LIN {X 0,Y 69.281,Z 314.928,A -85,B 0,C 180,E1 -28344.379,E2 -28344.379} C_VEL
LIN {X 0,Y 66.188,Z 315.169,A -85,B 0,C 180,E1 -28352.361,E2 -28352.361} C_VEL
LIN {X 0,Y 64.354,Z 314.872,A -85,B 0,C 180,E1 -28359.206,E2 -28359.206} C_VEL
LIN {X 0,Y 64.263,Z 314.308,A -85,B 0,C 180,E1 -28364.501,E2 -28364.501} C_VEL
LIN {X 0,Y 64.59,Z 313.988,A -85,B 0,C 180,E1 -28366.232,E2 -28366.232} C_VEL
LIN {X 0,Y 67.401,Z 312.213,A -85,B 0,C 180,E1 -28374.652,E2 -28374.652} C_VEL
LIN {X 0,Y 71.651,Z 309.343,A -85,B 0,C 180,E1 -28382.65,E2 -28382.65} C_VEL
LIN {X 0,Y 77.01,Z 305.448,A -85,B 0,C 180,E1 -28389.706,E2 -28389.706} C_VEL
LIN {X 0,Y 83.494,Z 300.415,A -85,B 0,C 180,E1 -28395.684,E2 -28395.684} C_VEL
LIN {X 0,Y 90.633,Z 294.076,A -85,B 0,C 180,E1 -28400.846,E2 -28400.846} C_VEL
LIN {X 0,Y 98.27,Z 286.156,A -85,B 0,C 180,E1 -28405.328,E2 -28405.328} C_VEL
LIN {X 0,Y 99.207,Z 284.697,A -85,B 0,C 180,E1 -28406.345,E2 -28406.345} C_VEL
LIN {X 0,Y 99.897,Z 283.172,A -85,B 0,C 180,E1 -28407.591,E2 -28407.591} C_VEL
LIN {X 0,Y 100.76,Z 279.934,A -85,B 0,C 180,E1 -28410.774,E2 -28410.774} C_VEL
LIN {X 0,Y 101.285,Z 275.871,A -85,B 0,C 180,E1 -28415.397,E2 -28415.397} C_VEL
LIN {X 0,Y 101.239,Z 272.91,A -85,B 0,C 180,E1 -28419.69,E2 -28419.69} C_VEL
LIN {X 0,Y 100.997,Z 270.647,A -85,B 0,C 180,E1 -28423.838,E2 -28423.838} C_VEL
LIN {X 0,Y 100.854,Z 268.882,A -85,B 0,C 180,E1 -28427.933,E2 -28427.933} C_VEL
LIN {X 0,Y 100.705,Z 267.66,A -85,B 0,C 180,E1 -28431.976,E2 -28431.976} C_VEL
LIN {X 0,Y 101.085,Z 266.25,A -85,B 0,C 180,E1 -28440,E2 -28440} C_VEL
LIN {X 0,Y 100.934,Z 268.18,A -85,B 0,C 180,E1 -28448.005,E2 -28448.005} C_VEL
LIN {X 0,Y 100.985,Z 270.458,A -85,B 0,C 180,E1 -28453.009,E2 -28453.009} C_VEL
LIN {X 0,Y 100.891,Z 273.868,A -85,B 0,C 180,E1 -28458.268,E2 -28458.268} C_VEL
LIN {X 0,Y 100.543,Z 277.522,A -85,B 0,C 180,E1 -28462.697,E2 -28462.697} C_VEL
LIN {X 0,Y 99.953,Z 281.758,A -85,B 0,C 180,E1 -28467.196,E2 -28467.196} C_VEL
LIN {X 0,Y 99.479,Z 284.247,A -85,B 0,C 180,E1 -28469.639,E2 -28469.639} C_VEL
LIN {X 0,Y 96.47,Z 289.372,A -85,B 0,C 180,E1 -28473.09,E2 -28473.09} C_VEL
LIN {X 0,Y 94.491,Z 292.269,A -85,B 0,C 180,E1 -28475.098,E2 -28475.098} C_VEL
LIN {X 0,Y 86.974,Z 299.696,A -85,B 0,C 180,E1 -28479.855,E2 -28479.855} C_VEL
LIN {X 0,Y 80.178,Z 305.666,A -85,B 0,C 180,E1 -28485.472,E2 -28485.472} C_VEL
LIN {X 0,Y 74.049,Z 310.379,A -85,B 0,C 180,E1 -28491.907,E2 -28491.907} C_VEL
LIN {X 0,Y 69,Z 313.984,A -85,B 0,C 180,E1 -28499.383,E2 -28499.383} C_VEL
LIN {X 0,Y 66.446,Z 315.847,A -85,B 0,C 180,E1 -28504.969,E2 -28504.969} C_VEL
LIN {X 0,Y 63.235,Z 318.251,A -85,B 0,C 180,E1 -28517.155,E2 -28517.155} C_VEL
LIN {X 0,Y 62.585,Z 318.865,A -85,B 0,C 180,E1 -28523.551,E2 -28523.551} C_VEL
LIN {X 0,Y 62.61,Z 319.084,A -85,B 0,C 180,E1 -28529.998,E2 -28529.998} C_VEL
LIN {X 0,Y 62.585,Z 318.848,A -85,B 0,C 180,E1 -28536.446,E2 -28536.446} C_VEL
LIN {X 0,Y 63.234,Z 318.224,A -85,B 0,C 180,E1 -28542.842,E2 -28542.842} C_VEL
LIN {X 0,Y 64.514,Z 317.21,A -85,B 0,C 180,E1 -28549.074,E2 -28549.074} C_VEL
LIN {X 0,Y 66.444,Z 315.792,A -85,B 0,C 180,E1 -28555.028,E2 -28555.028} C_VEL
LIN {X 0,Y 70.564,Z 312.831,A -85,B 0,C 180,E1 -28563.213,E2 -28563.213} C_VEL
LIN {X 0,Y 75.928,Z 308.835,A -85,B 0,C 180,E1 -28570.384,E2 -28570.384} C_VEL
LIN {X 0,Y 82.316,Z 303.761,A -85,B 0,C 180,E1 -28576.419,E2 -28576.419} C_VEL
LIN {X 0,Y 89.407,Z 297.236,A -85,B 0,C 180,E1 -28581.817,E2 -28581.817} C_VEL
LIN {X 0,Y 94.478,Z 292.065,A -85,B 0,C 180,E1 -28584.909,E2 -28584.909} C_VEL
LIN {X 0,Y 98.362,Z 286.011,A -85,B 0,C 180,E1 -28589.024,E2 -28589.024} C_VEL
LIN {X 0,Y 99.375,Z 284.107,A -85,B 0,C 180,E1 -28590.327,E2 -28590.327} C_VEL
LIN {X 0,Y 100.293,Z 278.836,A -85,B 0,C 180,E1 -28595.638,E2 -28595.638} C_VEL
LIN {X 0,Y 100.658,Z 275.358,A -85,B 0,C 180,E1 -28599.568,E2 -28599.568} C_VEL
LIN {X 0,Y 100.795,Z 273.641,A -85,B 0,C 180,E1 -28601.714,E2 -28601.714} C_VEL
LIN {X 0,Y 100.867,Z 269.735,A -85,B 0,C 180,E1 -28607.935,E2 -28607.935} C_VEL
LIN {X 0,Y 100.801,Z 267.955,A -85,B 0,C 180,E1 -28611.985,E2 -28611.985} C_VEL
LIN {X 0,Y 100.999,Z 265.946,A -85,B 0,C 180,E1 -28620,E2 -28620} C_VEL
LIN {X 0,Y 100.537,Z 267.452,A -85,B 0,C 180,E1 -28628.037,E2 -28628.037} C_VEL
LIN {X 0,Y 100.678,Z 268.755,A -85,B 0,C 180,E1 -28632.239,E2 -28632.239} C_VEL
LIN {X 0,Y 100.972,Z 271.484,A -85,B 0,C 180,E1 -28638.253,E2 -28638.253} C_VEL
LIN {X 0,Y 101.162,Z 274.398,A -85,B 0,C 180,E1 -28642.97,E2 -28642.97} C_VEL
LIN {X 0,Y 100.959,Z 277.552,A -85,B 0,C 180,E1 -28646.901,E2 -28646.901} C_VEL
LIN {X 0,Y 100.4,Z 281.102,A -85,B 0,C 180,E1 -28650.746,E2 -28650.746} C_VEL
LIN {X 0,Y 99.192,Z 284.396,A -85,B 0,C 180,E1 -28653.646,E2 -28653.646} C_VEL
LIN {X 0,Y 98.279,Z 285.853,A -85,B 0,C 180,E1 -28654.683,E2 -28654.683} C_VEL
LIN {X 0,Y 90.667,Z 293.824,A -85,B 0,C 180,E1 -28659.184,E2 -28659.184} C_VEL
LIN {X 0,Y 83.545,Z 300.222,A -85,B 0,C 180,E1 -28664.356,E2 -28664.356} C_VEL
LIN {X 0,Y 77.07,Z 305.298,A -85,B 0,C 180,E1 -28670.334,E2 -28670.334} C_VEL
LIN {X 0,Y 71.687,Z 309.231,A -85,B 0,C 180,E1 -28677.372,E2 -28677.372} C_VEL
LIN {X 0,Y 67.418,Z 312.134,A -85,B 0,C 180,E1 -28685.358,E2 -28685.358} C_VEL
LIN {X 0,Y 65.321,Z 313.516,A -85,B 0,C 180,E1 -28691.171,E2 -28691.171} C_VEL
LIN {X 0,Y 63.559,Z 314.641,A -85,B 0,C 180,E1 -28698.761,E2 -28698.761} C_VEL
LIN {X 0,Y 62.755,Z 315.321,A -85,B 0,C 180,E1 -28710.002,E2 -28710.002} C_VEL
LIN {X 0,Y 62.952,Z 315.125,A -85,B 0,C 180,E1 -28716.411,E2 -28716.411} C_VEL
LIN {X 0,Y 64.59,Z 313.988,A -85,B 0,C 180,E1 -28726.232,E2 -28726.232} C_VEL
LIN {X 0,Y 65.433,Z 313.116,A -85,B 0,C 180,E1 -28731.326,E2 -28731.326} C_VEL
LIN {X 0,Y 66.073,Z 311.171,A -85,B 0,C 180,E1 -28739.797,E2 -28739.797} C_VEL
LIN {X 0,Y 67.331,Z 309.128,A -85,B 0,C 180,E1 -28746.33,E2 -28746.33} C_VEL
LIN {X 0,Y 69.435,Z 307.235,A -85,B 0,C 180,E1 -28750.695,E2 -28750.695} C_VEL
LIN {X 0,Y 70.429,Z 306.505,A -85,B 0,C 180,E1 -28751.967,E2 -28751.967} C_VEL
LIN {X 0,Y 78.695,Z 300.627,A -85,B 0,C 180,E1 -28759.387,E2 -28759.387} C_VEL
LIN {X 0,Y 86.318,Z 294.288,A -85,B 0,C 180,E1 -28764.51,E2 -28764.51} C_VEL
LIN {X 0,Y 93.04,Z 287.838,A -85,B 0,C 180,E1 -28768.187,E2 -28768.187} C_VEL
LIN {X 0,Y 94.084,Z 286.385,A -85,B 0,C 180,E1 -28769.206,E2 -28769.206} C_VEL
LIN {X 0,Y 95.21,Z 283.449,A -85,B 0,C 180,E1 -28772.351,E2 -28772.351} C_VEL
LIN {X 0,Y 95.93,Z 280.382,A -85,B 0,C 180,E1 -28776.238,E2 -28776.238} C_VEL
LIN {X 0,Y 96.102,Z 278.815,A -85,B 0,C 180,E1 -28778.552,E2 -28778.552} C_VEL
LIN {X 0,Y 96.171,Z 276.419,A -85,B 0,C 180,E1 -28783.003,E2 -28783.003} C_VEL
LIN {X 0,Y 96.142,Z 274.594,A -85,B 0,C 180,E1 -28787.332,E2 -28787.332} C_VEL
LIN {X 0,Y 96.163,Z 273.324,A -85,B 0,C 180,E1 -28791.595,E2 -28791.595} C_VEL
LIN {X 0,Y 96.68,Z 271.872,A -85,B 0,C 180,E1 -28800,E2 -28800} C_VEL
LIN {X 0,Y 96.394,Z 272.739,A -85,B 0,C 180,E1 -28804.181,E2 -28804.181} C_VEL
LIN {X 0,Y 96.344,Z 273.942,A -85,B 0,C 180,E1 -28808.389,E2 -28808.389} C_VEL
LIN {X 0,Y 96.215,Z 275.756,A -85,B 0,C 180,E1 -28812.658,E2 -28812.658} C_VEL
LIN {X 0,Y 95.8,Z 278.757,A -85,B 0,C 180,E1 -28817.501,E2 -28817.501} C_VEL
LIN {X 0,Y 94.94,Z 283.03,A -85,B 0,C 180,E1 -28823.013,E2 -28823.013} C_VEL
LIN {X 0,Y 94.164,Z 286.139,A -85,B 0,C 180,E1 -28826.603,E2 -28826.603} C_VEL
LIN {X 0,Y 93.455,Z 287.742,A -85,B 0,C 180,E1 -28828.088,E2 -28828.088} C_VEL
LIN {X 0,Y 89.234,Z 293.419,A -85,B 0,C 180,E1 -28832.148,E2 -28832.148} C_VEL
LIN {X 0,Y 81.307,Z 300.599,A -85,B 0,C 180,E1 -28836.911,E2 -28836.911} C_VEL
LIN {X 0,Y 72.916,Z 307.143,A -85,B 0,C 180,E1 -28843.705,E2 -28843.705} C_VEL
LIN {X 0,Y 66.59,Z 311.475,A -85,B 0,C 180,E1 -28850.708,E2 -28850.708} C_VEL
LIN {X 0,Y 62.974,Z 313.771,A -85,B 0,C 180,E1 -28856.08,E2 -28856.08} C_VEL
LIN {X 0,Y 60.046,Z 315.633,A -85,B 0,C 180,E1 -28862.082,E2 -28862.082} C_VEL
LIN {X 0,Y 57.837,Z 317.035,A -85,B 0,C 180,E1 -28868.619,E2 -28868.619} C_VEL
LIN {X 0,Y 56.317,Z 318.038,A -85,B 0,C 180,E1 -28875.545,E2 -28875.545} C_VEL
LIN {X 0,Y 55.539,Z 318.652,A -85,B 0,C 180,E1 -28882.728,E2 -28882.728} C_VEL
LIN {X 0,Y 55.509,Z 318.871,A -85,B 0,C 180,E1 -28889.998,E2 -28889.998} C_VEL
LIN {X 0,Y 55.539,Z 318.635,A -85,B 0,C 180,E1 -28897.268,E2 -28897.268} C_VEL
LIN {X 0,Y 56.316,Z 318.01,A -85,B 0,C 180,E1 -28904.452,E2 -28904.452} C_VEL
LIN {X 0,Y 57.836,Z 316.996,A -85,B 0,C 180,E1 -28911.378,E2 -28911.378} C_VEL
LIN {X 0,Y 60.044,Z 315.577,A -85,B 0,C 180,E1 -28917.915,E2 -28917.915} C_VEL
LIN {X 0,Y 64.726,Z 312.617,A -85,B 0,C 180,E1 -28926.667,E2 -28926.667} C_VEL
LIN {X 0,Y 70.65,Z 308.62,A -85,B 0,C 180,E1 -28934.131,E2 -28934.131} C_VEL
LIN {X 0,Y 78.161,Z 303.03,A -85,B 0,C 180,E1 -28940.768,E2 -28940.768} C_VEL
LIN {X 0,Y 86.505,Z 295.781,A -85,B 0,C 180,E1 -28946.38,E2 -28946.38} C_VEL
LIN {X 0,Y 89.218,Z 293.211,A -85,B 0,C 180,E1 -28947.864,E2 -28947.864} C_VEL
LIN {X 0,Y 93.345,Z 287.598,A -85,B 0,C 180,E1 -28951.898,E2 -28951.898} C_VEL
LIN {X 0,Y 94.122,Z 285.742,A -85,B 0,C 180,E1 -28953.638,E2 -28953.638} C_VEL
LIN {X 0,Y 95.102,Z 281.697,A -85,B 0,C 180,E1 -28958.315,E2 -28958.315} C_VEL
LIN {X 0,Y 95.776,Z 278.217,A -85,B 0,C 180,E1 -28962.931,E2 -28962.931} C_VEL
LIN {X 0,Y 96.067,Z 275.596,A -85,B 0,C 180,E1 -28967.322,E2 -28967.322} C_VEL
LIN {X 0,Y 96.22,Z 273.733,A -85,B 0,C 180,E1 -28971.6,E2 -28971.6} C_VEL
LIN {X 0,Y 96.281,Z 272.503,A -85,B 0,C 180,E1 -28975.814,E2 -28975.814} C_VEL
LIN {X 0,Y 96.585,Z 271.605,A -85,B 0,C 180,E1 -28980,E2 -28980} C_VEL
LIN {X 0,Y 96.005,Z 273.131,A -85,B 0,C 180,E1 -28988.419,E2 -28988.419} C_VEL
LIN {X 0,Y 95.991,Z 274.397,A -85,B 0,C 180,E1 -28992.688,E2 -28992.688} C_VEL
LIN {X 0,Y 96.041,Z 276.672,A -85,B 0,C 180,E1 -28997.959,E2 -28997.959} C_VEL
LIN {X 0,Y 95.973,Z 278.608,A -85,B 0,C 180,E1 -29001.478,E2 -29001.478} C_VEL
LIN {X 0,Y 95.822,Z 280.153,A -85,B 0,C 180,E1 -29003.791,E2 -29003.791} C_VEL
LIN {X 0,Y 95.147,Z 283.132,A -85,B 0,C 180,E1 -29007.582,E2 -29007.582} C_VEL
LIN {X 0,Y 94.711,Z 284.658,A -85,B 0,C 180,E1 -29009.326,E2 -29009.326} C_VEL
LIN {X 0,Y 94.059,Z 286.09,A -85,B 0,C 180,E1 -29010.772,E2 -29010.772} C_VEL
LIN {X 0,Y 93.045,Z 287.546,A -85,B 0,C 180,E1 -29011.822,E2 -29011.822} C_VEL
LIN {X 0,Y 85.059,Z 295.201,A -85,B 0,C 180,E1 -29016.335,E2 -29016.335} C_VEL
LIN {X 0,Y 76.325,Z 302.242,A -85,B 0,C 180,E1 -29022.557,E2 -29022.557} C_VEL
LIN {X 0,Y 69.678,Z 306.925,A -85,B 0,C 180,E1 -29029.036,E2 -29029.036} C_VEL
LIN {X 0,Y 64.084,Z 310.502,A -85,B 0,C 180,E1 -29036.748,E2 -29036.748} C_VEL
LIN {X 0,Y 61.038,Z 312.347,A -85,B 0,C 180,E1 -29042.579,E2 -29042.579} C_VEL
LIN {X 0,Y 58.639,Z 313.729,A -85,B 0,C 180,E1 -29048.929,E2 -29048.929} C_VEL
LIN {X 0,Y 56.928,Z 314.712,A -85,B 0,C 180,E1 -29055.707,E2 -29055.707} C_VEL
LIN {X 0,Y 55.671,Z 315.534,A -85,B 0,C 180,E1 -29070.002,E2 -29070.002} C_VEL
LIN {X 0,Y 55.92,Z 315.337,A -85,B 0,C 180,E1 -29077.222,E2 -29077.222} C_VEL
LIN {X 0,Y 57.697,Z 314.258,A -85,B 0,C 180,E1 -29087.799,E2 -29087.799} C_VEL
LIN {X 0,Y 61.02,Z 312.425,A -85,B 0,C 180,E1 -29097.434,E2 -29097.434} C_VEL
LIN {X 0,Y 65.779,Z 309.555,A -85,B 0,C 180,E1 -29105.991,E2 -29105.991} C_VEL
LIN {X 0,Y 70.429,Z 306.505,A -85,B 0,C 180,E1 -29111.967,E2 -29111.967} C_VEL
LIN {X 0,Y 73.248,Z 304.257,A -85,B 0,C 180,E1 -29115.717,E2 -29115.717} C_VEL
LIN {X 0,Y 77.083,Z 300.21,A -85,B 0,C 180,E1 -29121.997,E2 -29121.997} C_VEL
LIN {X 0,Y 81.476,Z 295.53,A -85,B 0,C 180,E1 -29127.466,E2 -29127.466} C_VEL
LIN {X 0,Y 84.961,Z 292.254,A -85,B 0,C 180,E1 -29129.866,E2 -29129.866} C_VEL
LIN {X 0,Y 88.204,Z 289.28,A -85,B 0,C 180,E1 -29131.44,E2 -29131.44} C_VEL
LIN {X 0,Y 89.039,Z 288.193,A -85,B 0,C 180,E1 -29132.405,E2 -29132.405} C_VEL
LIN {X 0,Y 90.369,Z 284.706,A -85,B 0,C 180,E1 -29137.117,E2 -29137.117} C_VEL
LIN {X 0,Y 90.915,Z 281.96,A -85,B 0,C 180,E1 -29141.988,E2 -29141.988} C_VEL
LIN {X 0,Y 91.084,Z 280.079,A -85,B 0,C 180,E1 -29146.616,E2 -29146.616} C_VEL
LIN {X 0,Y 91.256,Z 278.71,A -85,B 0,C 180,E1 -29151.139,E2 -29151.139} C_VEL
LIN {X 0,Y 91.955,Z 277.266,A -85,B 0,C 180,E1 -29160,E2 -29160} C_VEL
LIN {X 0,Y 91.602,Z 278.147,A -85,B 0,C 180,E1 -29164.4,E2 -29164.4} C_VEL
LIN {X 0,Y 91.216,Z 280.312,A -85,B 0,C 180,E1 -29171.105,E2 -29171.105} C_VEL
LIN {X 0,Y 90.683,Z 282.756,A -85,B 0,C 180,E1 -29175.739,E2 -29175.739} C_VEL
LIN {X 0,Y 89.761,Z 285.668,A -85,B 0,C 180,E1 -29180.02,E2 -29180.02} C_VEL
LIN {X 0,Y 88.953,Z 288.097,A -85,B 0,C 180,E1 -29183.268,E2 -29183.268} C_VEL
LIN {X 0,Y 88.357,Z 289.564,A -85,B 0,C 180,E1 -29185.027,E2 -29185.027} C_VEL
LIN {X 0,Y 85.492,Z 293.197,A -85,B 0,C 180,E1 -29187.903,E2 -29187.903} C_VEL
LIN {X 0,Y 82.787,Z 295.758,A -85,B 0,C 180,E1 -29189.522,E2 -29189.522} C_VEL
LIN {X 0,Y 74.479,Z 302.483,A -85,B 0,C 180,E1 -29194.484,E2 -29194.484} C_VEL
LIN {X 0,Y 68.195,Z 306.931,A -85,B 0,C 180,E1 -29199.38,E2 -29199.38} C_VEL
LIN {X 0,Y 61.247,Z 311.262,A -85,B 0,C 180,E1 -29206.488,E2 -29206.488} C_VEL
LIN {X 0,Y 57.205,Z 313.558,A -85,B 0,C 180,E1 -29212.098,E2 -29212.098} C_VEL
LIN {X 0,Y 53.836,Z 315.419,A -85,B 0,C 180,E1 -29218.52,E2 -29218.52} C_VEL
LIN {X 0,Y 49.466,Z 317.825,A -85,B 0,C 180,E1 -29233.49,E2 -29233.49} C_VEL
LIN {X 0,Y 48.497,Z 318.439,A -85,B 0,C 180,E1 -29241.666,E2 -29241.666} C_VEL
LIN {X 0,Y 48.427,Z 318.658,A -85,B 0,C 180,E1 -29249.998,E2 -29249.998} C_VEL
LIN {X 0,Y 48.496,Z 318.421,A -85,B 0,C 180,E1 -29258.33,E2 -29258.33} C_VEL
LIN {X 0,Y 49.465,Z 317.796,A -85,B 0,C 180,E1 -29266.506,E2 -29266.506} C_VEL
LIN {X 0,Y 51.249,Z 316.781,A -85,B 0,C 180,E1 -29274.291,E2 -29274.291} C_VEL
LIN {X 0,Y 53.834,Z 315.361,A -85,B 0,C 180,E1 -29281.477,E2 -29281.477} C_VEL
LIN {X 0,Y 59.172,Z 312.402,A -85,B 0,C 180,E1 -29290.785,E2 -29290.785} C_VEL
LIN {X 0,Y 65.727,Z 308.405,A -85,B 0,C 180,E1 -29298.457,E2 -29298.457} C_VEL
LIN {X 0,Y 74.335,Z 302.424,A -85,B 0,C 180,E1 -29305.44,E2 -29305.44} C_VEL
LIN {X 0,Y 82.774,Z 295.565,A -85,B 0,C 180,E1 -29310.488,E2 -29310.488} C_VEL
LIN {X 0,Y 85.477,Z 292.984,A -85,B 0,C 180,E1 -29312.11,E2 -29312.11} C_VEL
LIN {X 0,Y 88.245,Z 289.43,A -85,B 0,C 180,E1 -29314.939,E2 -29314.939} C_VEL
LIN {X 0,Y 89.717,Z 285.402,A -85,B 0,C 180,E1 -29320.052,E2 -29320.052} C_VEL
LIN {X 0,Y 90.599,Z 282.56,A -85,B 0,C 180,E1 -29324.246,E2 -29324.246} C_VEL
LIN {X 0,Y 91.092,Z 280.138,A -85,B 0,C 180,E1 -29328.879,E2 -29328.879} C_VEL
LIN {X 0,Y 91.497,Z 277.935,A -85,B 0,C 180,E1 -29335.595,E2 -29335.595} C_VEL
LIN {X 0,Y 91.869,Z 277.014,A -85,B 0,C 180,E1 -29340,E2 -29340} C_VEL
LIN {X 0,Y 91.139,Z 278.277,A -85,B 0,C 180,E1 -29347.672,E2 -29347.672} C_VEL
LIN {X 0,Y 90.952,Z 279.882,A -85,B 0,C 180,E1 -29353.404,E2 -29353.404} C_VEL
LIN {X 0,Y 90.762,Z 281.797,A -85,B 0,C 180,E1 -29358.043,E2 -29358.043} C_VEL
LIN {X 0,Y 90.273,Z 284.494,A -85,B 0,C 180,E1 -29362.909,E2 -29362.909} C_VEL
LIN {X 0,Y 89.019,Z 287.913,A -85,B 0,C 180,E1 -29367.575,E2 -29367.575} C_VEL
LIN {X 0,Y 88.078,Z 289.136,A -85,B 0,C 180,E1 -29368.634,E2 -29368.634} C_VEL
LIN {X 0,Y 79.7,Z 296.524,A -85,B 0,C 180,E1 -29373.102,E2 -29373.102} C_VEL
LIN {X 0,Y 71.708,Z 302.457,A -85,B 0,C 180,E1 -29378.368,E2 -29378.368} C_VEL
LIN {X 0,Y 64.466,Z 307.14,A -85,B 0,C 180,E1 -29384.88,E2 -29384.88} C_VEL
LIN {X 0,Y 58.264,Z 310.717,A -85,B 0,C 180,E1 -29392.909,E2 -29392.909} C_VEL
LIN {X 0,Y 54.84,Z 312.561,A -85,B 0,C 180,E1 -29399.164,E2 -29399.164} C_VEL
LIN {X 0,Y 52.08,Z 313.943,A -85,B 0,C 180,E1 -29406.121,E2 -29406.121} C_VEL
LIN {X 0,Y 50.086,Z 314.925,A -85,B 0,C 180,E1 -29413.704,E2 -29413.704} C_VEL
LIN {X 0,Y 48.581,Z 315.746,A -85,B 0,C 180,E1 -29430.002,E2 -29430.002} C_VEL
LIN {X 0,Y 48.885,Z 315.55,A -85,B 0,C 180,E1 -29438.268,E2 -29438.268} C_VEL
LIN {X 0,Y 50.086,Z 314.963,A -85,B 0,C 180,E1 -29446.3,E2 -29446.3} C_VEL
LIN {X 0,Y 54.822,Z 312.638,A -85,B 0,C 180,E1 -29460.851,E2 -29460.851} C_VEL
LIN {X 0,Y 60.176,Z 309.767,A -85,B 0,C 180,E1 -29469.969,E2 -29469.969} C_VEL
LIN {X 0,Y 66.696,Z 305.873,A -85,B 0,C 180,E1 -29477.53,E2 -29477.53} C_VEL
LIN {X 0,Y 74.268,Z 300.839,A -85,B 0,C 180,E1 -29483.551,E2 -29483.551} C_VEL
LIN {X 0,Y 82.393,Z 294.499,A -85,B 0,C 180,E1 -29488.539,E2 -29488.539} C_VEL
LIN {X 0,Y 84.961,Z 292.254,A -85,B 0,C 180,E1 -29489.866,E2 -29489.866} C_VEL
LIN {X 0,Y 86.403,Z 290.598,A -85,B 0,C 180,E1 -29491.316,E2 -29491.316} C_VEL
LIN {X 0,Y 86.918,Z 289.295,A -85,B 0,C 180,E1 -29493.231,E2 -29493.231} C_VEL
LIN {X 0,Y 86.766,Z 288.216,A -85,B 0,C 180,E1 -29495.751,E2 -29495.751} C_VEL
LIN {X 0,Y 85.514,Z 286.072,A -85,B 0,C 180,E1 -29503.595,E2 -29503.595} C_VEL
LIN {X 0,Y 86.013,Z 283.861,A -85,B 0,C 180,E1 -29510.594,E2 -29510.594} C_VEL
LIN {X 0,Y 86.354,Z 282.947,A -85,B 0,C 180,E1 -29515.332,E2 -29515.332} C_VEL
LIN {X 0,Y 86.921,Z 282.366,A -85,B 0,C 180,E1 -29520,E2 -29520} C_VEL
LIN {X 0,Y 86.449,Z 283.276,A -85,B 0,C 180,E1 -29524.663,E2 -29524.663} C_VEL
LIN {X 0,Y 85.871,Z 285.236,A -85,B 0,C 180,E1 -29530.843,E2 -29530.843} C_VEL
LIN {X 0,Y 85.33,Z 286.863,A -85,B 0,C 180,E1 -29534.305,E2 -29534.305} C_VEL
LIN {X 0,Y 83.877,Z 290.158,A -85,B 0,C 180,E1 -29539.582,E2 -29539.582} C_VEL
LIN {X 0,Y 83.2,Z 291.569,A -85,B 0,C 180,E1 -29541.689,E2 -29541.689} C_VEL
LIN {X 0,Y 82.157,Z 292.968,A -85,B 0,C 180,E1 -29543.131,E2 -29543.131} C_VEL
LIN {X 0,Y 80.918,Z 294.302,A -85,B 0,C 180,E1 -29544.22,E2 -29544.22} C_VEL
LIN {X 0,Y 73.608,Z 300.173,A -85,B 0,C 180,E1 -29547.969,E2 -29547.969} C_VEL
LIN {X 0,Y 63.917,Z 306.719,A -85,B 0,C 180,E1 -29554.443,E2 -29554.443} C_VEL
LIN {X 0,Y 56.299,Z 311.049,A -85,B 0,C 180,E1 -29561.493,E2 -29561.493} C_VEL
LIN {X 0,Y 51.778,Z 313.345,A -85,B 0,C 180,E1 -29567.258,E2 -29567.258} C_VEL
LIN {X 0,Y 47.891,Z 315.206,A -85,B 0,C 180,E1 -29574.053,E2 -29574.053} C_VEL
LIN {X 0,Y 42.675,Z 317.611,A -85,B 0,C 180,E1 -29590.767,E2 -29590.767} C_VEL
LIN {X 0,Y 41.471,Z 318.226,A -85,B 0,C 180,E1 -29600.241,E2 -29600.241} C_VEL
LIN {X 0,Y 41.327,Z 318.445,A -85,B 0,C 180,E1 -29609.998,E2 -29609.998} C_VEL
LIN {X 0,Y 41.47,Z 318.208,A -85,B 0,C 180,E1 -29619.755,E2 -29619.755} C_VEL
LIN {X 0,Y 42.674,Z 317.582,A -85,B 0,C 180,E1 -29629.229,E2 -29629.229} C_VEL
LIN {X 0,Y 44.835,Z 316.566,A -85,B 0,C 180,E1 -29638.049,E2 -29638.049} C_VEL
LIN {X 0,Y 47.889,Z 315.146,A -85,B 0,C 180,E1 -29645.944,E2 -29645.944} C_VEL
LIN {X 0,Y 53.967,Z 312.187,A -85,B 0,C 180,E1 -29655.743,E2 -29655.743} C_VEL
LIN {X 0,Y 61.24,Z 308.19,A -85,B 0,C 180,E1 -29663.447,E2 -29663.447} C_VEL
LIN {X 0,Y 69.904,Z 302.663,A -85,B 0,C 180,E1 -29669.822,E2 -29669.822} C_VEL
LIN {X 0,Y 79.502,Z 295.349,A -85,B 0,C 180,E1 -29674.968,E2 -29674.968} C_VEL
LIN {X 0,Y 80.904,Z 294.104,A -85,B 0,C 180,E1 -29675.796,E2 -29675.796} C_VEL
LIN {X 0,Y 82.144,Z 292.749,A -85,B 0,C 180,E1 -29676.885,E2 -29676.885} C_VEL
LIN {X 0,Y 83.134,Z 291.345,A -85,B 0,C 180,E1 -29678.418,E2 -29678.418} C_VEL
LIN {X 0,Y 84.573,Z 288.214,A -85,B 0,C 180,E1 -29683.091,E2 -29683.091} C_VEL
LIN {X 0,Y 85.238,Z 286.694,A -85,B 0,C 180,E1 -29685.679,E2 -29685.679} C_VEL
LIN {X 0,Y 85.946,Z 284.477,A -85,B 0,C 180,E1 -29690.588,E2 -29690.588} C_VEL
LIN {X 0,Y 86.345,Z 283.088,A -85,B 0,C 180,E1 -29695.331,E2 -29695.331} C_VEL
LIN {X 0,Y 86.864,Z 282.129,A -85,B 0,C 180,E1 -29700,E2 -29700} C_VEL
LIN {X 0,Y 86.288,Z 282.714,A -85,B 0,C 180,E1 -29704.672,E2 -29704.672} C_VEL
LIN {X 0,Y 85.801,Z 283.991,A -85,B 0,C 180,E1 -29710.611,E2 -29710.611} C_VEL
LIN {X 0,Y 85.357,Z 286.027,A -85,B 0,C 180,E1 -29716.749,E2 -29716.749} C_VEL
LIN {X 0,Y 84.781,Z 288.07,A -85,B 0,C 180,E1 -29721.08,E2 -29721.08} C_VEL
LIN {X 0,Y 83.606,Z 290.463,A -85,B 0,C 180,E1 -29724.854,E2 -29724.854} C_VEL
LIN {X 0,Y 74.618,Z 297.848,A -85,B 0,C 180,E1 -29729.402,E2 -29729.402} C_VEL
LIN {X 0,Y 67.528,Z 302.672,A -85,B 0,C 180,E1 -29733.636,E2 -29733.636} C_VEL
LIN {X 0,Y 59.658,Z 307.355,A -85,B 0,C 180,E1 -29740.031,E2 -29740.031} C_VEL
LIN {X 0,Y 52.77,Z 310.931,A -85,B 0,C 180,E1 -29748.25,E2 -29748.25} C_VEL
LIN {X 0,Y 48.878,Z 312.775,A -85,B 0,C 180,E1 -29754.893,E2 -29754.893} C_VEL
LIN {X 0,Y 43.336,Z 315.138,A -85,B 0,C 180,E1 -29771.076,E2 -29771.076} C_VEL
LIN {X 0,Y 41.481,Z 315.959,A -85,B 0,C 180,E1 -29790.002,E2 -29790.002} C_VEL
LIN {X 0,Y 41.888,Z 315.762,A -85,B 0,C 180,E1 -29799.661,E2 -29799.661} C_VEL
LIN {X 0,Y 43.336,Z 315.175,A -85,B 0,C 180,E1 -29808.929,E2 -29808.929} C_VEL
LIN {X 0,Y 48.848,Z 312.851,A -85,B 0,C 180,E1 -29825.137,E2 -29825.137} C_VEL
LIN {X 0,Y 54.923,Z 309.979,A -85,B 0,C 180,E1 -29834.734,E2 -29834.734} C_VEL
LIN {X 0,Y 62.125,Z 306.084,A -85,B 0,C 180,E1 -29842.364,E2 -29842.364} C_VEL
LIN {X 0,Y 70.282,Z 301.05,A -85,B 0,C 180,E1 -29848.211,E2 -29848.211} C_VEL
LIN {X 0,Y 78.919,Z 294.71,A -85,B 0,C 180,E1 -29852.942,E2 -29852.942} C_VEL
LIN {X 0,Y 83.648,Z 290.692,A -85,B 0,C 180,E1 -29855.159,E2 -29855.159} C_VEL
LIN {X 0,Y 84.844,Z 288.364,A -85,B 0,C 180,E1 -29858.769,E2 -29858.769} C_VEL
LIN {X 0,Y 85.514,Z 286.072,A -85,B 0,C 180,E1 -29863.595,E2 -29863.595} C_VEL
LIN {X 0,Y 85.266,Z 285.206,A -85,B 0,C 180,E1 -29867.544,E2 -29867.544} C_VEL
LIN {X 0,Y 84.458,Z 285.145,A -85,B 0,C 180,E1 -29871.551,E2 -29871.551} C_VEL
LIN {X 0,Y 82.963,Z 285.971,A -85,B 0,C 180,E1 -29876.98,E2 -29876.98} C_VEL
LIN {X 0,Y 80.91,Z 288.258,A -85,B 0,C 180,E1 -29885.347,E2 -29885.347} C_VEL
LIN {X 0,Y 80.362,Z 289.661,A -85,B 0,C 180,E1 -29890.073,E2 -29890.073} C_VEL
LIN {X 0,Y 79.544,Z 291.212,A -85,B 0,C 180,E1 -29893.612,E2 -29893.612} C_VEL
LIN {X 0,Y 77.868,Z 294.054,A -85,B 0,C 180,E1 -29898.612,E2 -29898.612} C_VEL
LIN {X 0,Y 76.707,Z 295.329,A -85,B 0,C 180,E1 -29900.092,E2 -29900.092} C_VEL
LIN {X 0,Y 67.468,Z 302.029,A -85,B 0,C 180,E1 -29904.403,E2 -29904.403} C_VEL
LIN {X 0,Y 57.295,Z 308.093,A -85,B 0,C 180,E1 -29910.832,E2 -29910.832} C_VEL
LIN {X 0,Y 49.259,Z 312.058,A -85,B 0,C 180,E1 -29918.303,E2 -29918.303} C_VEL
LIN {X 0,Y 42.32,Z 314.992,A -85,B 0,C 180,E1 -29928.37,E2 -29928.37} C_VEL
LIN {X 0,Y 36.027,Z 317.398,A -85,B 0,C 180,E1 -29947.033,E2 -29947.033} C_VEL
LIN {X 0,Y 34.492,Z 318.013,A -85,B 0,C 180,E1 -29958.24,E2 -29958.24} C_VEL
LIN {X 0,Y 34.242,Z 318.232,A -85,B 0,C 180,E1 -29969.997,E2 -29969.997} C_VEL
LIN {X 0,Y 34.492,Z 317.994,A -85,B 0,C 180,E1 -29981.754,E2 -29981.754} C_VEL
LIN {X 0,Y 36.026,Z 317.367,A -85,B 0,C 180,E1 -29992.962,E2 -29992.962} C_VEL
LIN {X 0,Y 38.685,Z 316.351,A -85,B 0,C 180,E1 -30003.023,E2 -30003.023} C_VEL
LIN {X 0,Y 42.317,Z 314.931,A -85,B 0,C 180,E1 -30011.627,E2 -30011.627} C_VEL
LIN {X 0,Y 49.256,Z 311.972,A -85,B 0,C 180,E1 -30021.695,E2 -30021.695} C_VEL
LIN {X 0,Y 57.29,Z 307.975,A -85,B 0,C 180,E1 -30029.17,E2 -30029.17} C_VEL
LIN {X 0,Y 66.634,Z 302.426,A -85,B 0,C 180,E1 -30035.152,E2 -30035.152} C_VEL
LIN {X 0,Y 76.702,Z 295.128,A -85,B 0,C 180,E1 -30039.909,E2 -30039.909} C_VEL
LIN {X 0,Y 77.828,Z 293.848,A -85,B 0,C 180,E1 -30041.467,E2 -30041.467} C_VEL
LIN {X 0,Y 79.498,Z 290.98,A -85,B 0,C 180,E1 -30046.513,E2 -30046.513} C_VEL
LIN {X 0,Y 80.253,Z 289.503,A -85,B 0,C 180,E1 -30049.913,E2 -30049.913} C_VEL
LIN {X 0,Y 80.877,Z 287.973,A -85,B 0,C 180,E1 -30055.015,E2 -30055.015} C_VEL
LIN {X 0,Y 81.527,Z 286.951,A -85,B 0,C 180,E1 -30060,E2 -30060} C_VEL
LIN {X 0,Y 80.585,Z 287.982,A -85,B 0,C 180,E1 -30067.247,E2 -30067.247} C_VEL
LIN {X 0,Y 80.387,Z 288.534,A -85,B 0,C 180,E1 -30070.07,E2 -30070.07} C_VEL
LIN {X 0,Y 79.817,Z 290.027,A -85,B 0,C 180,E1 -30075.317,E2 -30075.317} C_VEL
LIN {X 0,Y 79.407,Z 291.061,A -85,B 0,C 180,E1 -30078.046,E2 -30078.046} C_VEL
LIN {X 0,Y 78.643,Z 292.489,A -85,B 0,C 180,E1 -30080.945,E2 -30080.945} C_VEL
LIN {X 0,Y 75.969,Z 294.686,A -85,B 0,C 180,E1 -30082.319,E2 -30082.319} C_VEL
LIN {X 0,Y 66.846,Z 301.081,A -85,B 0,C 180,E1 -30086.666,E2 -30086.666} C_VEL
LIN {X 0,Y 58.096,Z 306.156,A -85,B 0,C 180,E1 -30092.137,E2 -30092.137} C_VEL
LIN {X 0,Y 50.162,Z 310.088,A -85,B 0,C 180,E1 -30099.597,E2 -30099.597} C_VEL
LIN {X 0,Y 43.254,Z 312.989,A -85,B 0,C 180,E1 -30109.467,E2 -30109.467} C_VEL
LIN {X 0,Y 36.696,Z 315.351,A -85,B 0,C 180,E1 -30127.481,E2 -30127.481} C_VEL
LIN {X 0,Y 34.4,Z 316.172,A -85,B 0,C 180,E1 -30150.003,E2 -30150.003} C_VEL
LIN {X 0,Y 34.92,Z 315.975,A -85,B 0,C 180,E1 -30161.614,E2 -30161.614} C_VEL
LIN {X 0,Y 36.696,Z 315.388,A -85,B 0,C 180,E1 -30172.525,E2 -30172.525} C_VEL
LIN {X 0,Y 43.229,Z 313.063,A -85,B 0,C 180,E1 -30190.567,E2 -30190.567} C_VEL
LIN {X 0,Y 50.129,Z 310.192,A -85,B 0,C 180,E1 -30200.455,E2 -30200.455} C_VEL
LIN {X 0,Y 58.066,Z 306.296,A -85,B 0,C 180,E1 -30207.916,E2 -30207.916} C_VEL
LIN {X 0,Y 66.817,Z 301.261,A -85,B 0,C 180,E1 -30213.39,E2 -30213.39} C_VEL
LIN {X 0,Y 75.954,Z 294.921,A -85,B 0,C 180,E1 -30217.715,E2 -30217.715} C_VEL
LIN {X 0,Y 78.706,Z 292.677,A -85,B 0,C 180,E1 -30219.073,E2 -30219.073} C_VEL
LIN {X 0,Y 79.51,Z 291.235,A -85,B 0,C 180,E1 -30221.978,E2 -30221.978} C_VEL
LIN {X 0,Y 79.978,Z 290.048,A -85,B 0,C 180,E1 -30225.158,E2 -30225.158} C_VEL
LIN {X 0,Y 80.527,Z 288.688,A -85,B 0,C 180,E1 -30229.947,E2 -30229.947} C_VEL
LIN {X 0,Y 80.951,Z 287.753,A -85,B 0,C 180,E1 -30235.019,E2 -30235.019} C_VEL
LIN {X 0,Y 81.578,Z 287.172,A -85,B 0,C 180,E1 -30240,E2 -30240} C_VEL
LIN {X 0,Y 80.91,Z 288.258,A -85,B 0,C 180,E1 -30245.347,E2 -30245.347} C_VEL
LIN {X 0,Y 79.983,Z 289.522,A -85,B 0,C 180,E1 -30248.075,E2 -30248.075} C_VEL
LIN {X 0,Y 78.386,Z 291.295,A -85,B 0,C 180,E1 -30250.545,E2 -30250.545} C_VEL
LIN {X 0,Y 75.477,Z 294.106,A -85,B 0,C 180,E1 -30253.439,E2 -30253.439} C_VEL
LIN {X 0,Y 71.818,Z 297.137,A -85,B 0,C 180,E1 -30255.806,E2 -30255.806} C_VEL
LIN {X 0,Y 69.722,Z 298.627,A -85,B 0,C 180,E1 -30256.705,E2 -30256.705} C_VEL
LIN {X 0,Y 60.16,Z 304.6,A -85,B 0,C 180,E1 -30260.837,E2 -30260.837} C_VEL
LIN {X 0,Y 50.966,Z 309.314,A -85,B 0,C 180,E1 -30266.316,E2 -30266.316} C_VEL
LIN {X 0,Y 42.427,Z 312.919,A -85,B 0,C 180,E1 -30274.078,E2 -30274.078} C_VEL
LIN {X 0,Y 37.288,Z 314.779,A -85,B 0,C 180,E1 -30281.066,E2 -30281.066} C_VEL
LIN {X 0,Y 29.608,Z 317.184,A -85,B 0,C 180,E1 -30301.654,E2 -30301.654} C_VEL
LIN {X 0,Y 27.561,Z 317.8,A -85,B 0,C 180,E1 -30315.223,E2 -30315.223} C_VEL
LIN {X 0,Y 27.129,Z 318.019,A -85,B 0,C 180,E1 -30329.996,E2 -30329.996} C_VEL
LIN {X 0,Y 27.561,Z 317.781,A -85,B 0,C 180,E1 -30344.77,E2 -30344.77} C_VEL
LIN {X 0,Y 29.606,Z 317.154,A -85,B 0,C 180,E1 -30358.34,E2 -30358.34} C_VEL
LIN {X 0,Y 32.94,Z 316.137,A -85,B 0,C 180,E1 -30369.793,E2 -30369.793} C_VEL
LIN {X 0,Y 37.285,Z 314.717,A -85,B 0,C 180,E1 -30378.931,E2 -30378.931} C_VEL
LIN {X 0,Y 45.185,Z 311.757,A -85,B 0,C 180,E1 -30388.805,E2 -30388.805} C_VEL
LIN {X 0,Y 53.991,Z 307.761,A -85,B 0,C 180,E1 -30395.666,E2 -30395.666} C_VEL
LIN {X 0,Y 63.575,Z 302.459,A -85,B 0,C 180,E1 -30400.779,E2 -30400.779} C_VEL
LIN {X 0,Y 71.324,Z 297.326,A -85,B 0,C 180,E1 -30403.884,E2 -30403.884} C_VEL
LIN {X 0,Y 72.688,Z 296.123,A -85,B 0,C 180,E1 -30405.204,E2 -30405.204} C_VEL
LIN {X 0,Y 74.044,Z 294.292,A -85,B 0,C 180,E1 -30409.057,E2 -30409.057} C_VEL
LIN {X 0,Y 75.105,Z 292.58,A -85,B 0,C 180,E1 -30414.631,E2 -30414.631} C_VEL
LIN {X 0,Y 75.9,Z 291.5,A -85,B 0,C 180,E1 -30420,E2 -30420} C_VEL
LIN {X 0,Y 74.944,Z 292.353,A -85,B 0,C 180,E1 -30426.77,E2 -30426.77} C_VEL
LIN {X 0,Y 74.5,Z 293.114,A -85,B 0,C 180,E1 -30430.876,E2 -30430.876} C_VEL
LIN {X 0,Y 73.487,Z 294.91,A -85,B 0,C 180,E1 -30436.994,E2 -30436.994} C_VEL
LIN {X 0,Y 68.766,Z 298.278,A -85,B 0,C 180,E1 -30439.033,E2 -30439.033} C_VEL
LIN {X 0,Y 60.824,Z 303.101,A -85,B 0,C 180,E1 -30442.431,E2 -30442.431} C_VEL
LIN {X 0,Y 51.677,Z 307.784,A -85,B 0,C 180,E1 -30447.876,E2 -30447.876} C_VEL
LIN {X 0,Y 43.228,Z 311.359,A -85,B 0,C 180,E1 -30455.624,E2 -30455.624} C_VEL
LIN {X 0,Y 38.137,Z 313.203,A -85,B 0,C 180,E1 -30462.516,E2 -30462.516} C_VEL
LIN {X 0,Y 33.723,Z 314.584,A -85,B 0,C 180,E1 -30471.307,E2 -30471.307} C_VEL
LIN {X 0,Y 30.256,Z 315.565,A -85,B 0,C 180,E1 -30482.321,E2 -30482.321} C_VEL
LIN {X 0,Y 27.302,Z 316.385,A -85,B 0,C 180,E1 -30510.004,E2 -30510.004} C_VEL
LIN {X 0,Y 28,Z 316.188,A -85,B 0,C 180,E1 -30524.54,E2 -30524.54} C_VEL
LIN {X 0,Y 30.256,Z 315.601,A -85,B 0,C 180,E1 -30537.686,E2 -30537.686} C_VEL
LIN {X 0,Y 38.117,Z 313.276,A -85,B 0,C 180,E1 -30557.525,E2 -30557.525} C_VEL
LIN {X 0,Y 45.922,Z 310.405,A -85,B 0,C 180,E1 -30567.327,E2 -30567.327} C_VEL
LIN {X 0,Y 54.632,Z 306.508,A -85,B 0,C 180,E1 -30574.228,E2 -30574.228} C_VEL
LIN {X 0,Y 63.955,Z 301.473,A -85,B 0,C 180,E1 -30579.082,E2 -30579.082} C_VEL
LIN {X 0,Y 73.542,Z 295.133,A -85,B 0,C 180,E1 -30582.874,E2 -30582.874} C_VEL
LIN {X 0,Y 74.614,Z 293.26,A -85,B 0,C 180,E1 -30589.141,E2 -30589.141} C_VEL
LIN {X 0,Y 75.265,Z 292.275,A -85,B 0,C 180,E1 -30594.642,E2 -30594.642} C_VEL
LIN {X 0,Y 75.952,Z 291.702,A -85,B 0,C 180,E1 -30600,E2 -30600} C_VEL
LIN {X 0,Y 75.193,Z 292.748,A -85,B 0,C 180,E1 -30605.363,E2 -30605.363} C_VEL
LIN {X 0,Y 74.117,Z 294.45,A -85,B 0,C 180,E1 -30610.932,E2 -30610.932} C_VEL
LIN {X 0,Y 72.725,Z 296.332,A -85,B 0,C 180,E1 -30614.894,E2 -30614.894} C_VEL
LIN {X 0,Y 71.338,Z 297.513,A -85,B 0,C 180,E1 -30616.146,E2 -30616.146} C_VEL
LIN {X 0,Y 69.722,Z 298.627,A -85,B 0,C 180,E1 -30616.705,E2 -30616.705} C_VEL
LIN {X 0,Y 64.861,Z 301.68,A -85,B 0,C 180,E1 -30617.944,E2 -30617.944} C_VEL
LIN {X 0,Y 56.044,Z 306.137,A -85,B 0,C 180,E1 -30618.919,E2 -30618.919} C_VEL
LIN {X 0,Y 46.925,Z 309.844,A -85,B 0,C 180,E1 -30620.407,E2 -30620.407} C_VEL
LIN {X 0,Y 41.686,Z 311.721,A -85,B 0,C 180,E1 -30623.028,E2 -30623.028} C_VEL
LIN {X 0,Y 33.041,Z 314.565,A -85,B 0,C 180,E1 -30631.694,E2 -30631.694} C_VEL
LIN {X 0,Y 27.848,Z 315.967,A -85,B 0,C 180,E1 -30640.786,E2 -30640.786} C_VEL
LIN {X 0,Y 20.77,Z 317.587,A -85,B 0,C 180,E1 -30670.217,E2 -30670.217} C_VEL
LIN {X 0,Y 20.022,Z 317.806,A -85,B 0,C 180,E1 -30689.995,E2 -30689.995} C_VEL
LIN {X 0,Y 20.769,Z 317.567,A -85,B 0,C 180,E1 -30709.774,E2 -30709.774} C_VEL
LIN {X 0,Y 27.846,Z 315.923,A -85,B 0,C 180,E1 -30739.21,E2 -30739.21} C_VEL
LIN {X 0,Y 33.038,Z 314.502,A -85,B 0,C 180,E1 -30748.304,E2 -30748.304} C_VEL
LIN {X 0,Y 41.939,Z 311.542,A -85,B 0,C 180,E1 -30757.165,E2 -30757.165} C_VEL
LIN {X 0,Y 51.468,Z 307.546,A -85,B 0,C 180,E1 -30762.904,E2 -30762.904} C_VEL
LIN {X 0,Y 62.975,Z 301.402,A -85,B 0,C 180,E1 -30767.54,E2 -30767.54} C_VEL
LIN {X 0,Y 67.46,Z 298.59,A -85,B 0,C 180,E1 -30768.928,E2 -30768.928} C_VEL
LIN {X 0,Y 68.353,Z 297.626,A -85,B 0,C 180,E1 -30771.433,E2 -30771.433} C_VEL
LIN {X 0,Y 68.909,Z 296.922,A -85,B 0,C 180,E1 -30774.146,E2 -30774.146} C_VEL
LIN {X 0,Y 70.026,Z 295.737,A -85,B 0,C 180,E1 -30780,E2 -30780} C_VEL
LIN {X 0,Y 69.172,Z 296.333,A -85,B 0,C 180,E1 -30785.939,E2 -30785.939} C_VEL
LIN {X 0,Y 68.206,Z 297.431,A -85,B 0,C 180,E1 -30791.893,E2 -30791.893} C_VEL
LIN {X 0,Y 67.092,Z 298.287,A -85,B 0,C 180,E1 -30793.139,E2 -30793.139} C_VEL
LIN {X 0,Y 58.487,Z 303.315,A -85,B 0,C 180,E1 -30795.996,E2 -30795.996} C_VEL
LIN {X 0,Y 48.764,Z 307.998,A -85,B 0,C 180,E1 -30800.487,E2 -30800.487} C_VEL
LIN {X 0,Y 39.522,Z 311.573,A -85,B 0,C 180,E1 -30807.242,E2 -30807.242} C_VEL
LIN {X 0,Y 33.75,Z 313.416,A -85,B 0,C 180,E1 -30813.603,E2 -30813.603} C_VEL
LIN {X 0,Y 24.201,Z 315.778,A -85,B 0,C 180,E1 -30834.497,E2 -30834.497} C_VEL
LIN {X 0,Y 20.22,Z 316.598,A -85,B 0,C 180,E1 -30870.005,E2 -30870.005} C_VEL
LIN {X 0,Y 21.207,Z 316.401,A -85,B 0,C 180,E1 -30889.358,E2 -30889.358} C_VEL
LIN {X 0,Y 24.201,Z 315.813,A -85,B 0,C 180,E1 -30905.512,E2 -30905.512} C_VEL
LIN {X 0,Y 33.736,Z 313.488,A -85,B 0,C 180,E1 -30926.444,E2 -30926.444} C_VEL
LIN {X 0,Y 42.504,Z 310.617,A -85,B 0,C 180,E1 -30935.431,E2 -30935.431} C_VEL
LIN {X 0,Y 51.944,Z 306.719,A -85,B 0,C 180,E1 -30941.284,E2 -30941.284} C_VEL
LIN {X 0,Y 61.779,Z 301.684,A -85,B 0,C 180,E1 -30945.238,E2 -30945.238} C_VEL
LIN {X 0,Y 67.178,Z 298.424,A -85,B 0,C 180,E1 -30946.975,E2 -30946.975} C_VEL
LIN {X 0,Y 68.299,Z 297.576,A -85,B 0,C 180,E1 -30948.123,E2 -30948.123} C_VEL
LIN {X 0,Y 69.267,Z 296.469,A -85,B 0,C 180,E1 -30954.176,E2 -30954.176} C_VEL
LIN {X 0,Y 70.064,Z 295.927,A -85,B 0,C 180,E1 -30960,E2 -30960} C_VEL
LIN {X 0,Y 68.976,Z 297.073,A -85,B 0,C 180,E1 -30965.848,E2 -30965.848} C_VEL
LIN {X 0,Y 68.406,Z 297.784,A -85,B 0,C 180,E1 -30968.558,E2 -30968.558} C_VEL
LIN {X 0,Y 67.527,Z 298.729,A -85,B 0,C 180,E1 -30971.013,E2 -30971.013} C_VEL
LIN {X 0,Y 58.003,Z 304.387,A -85,B 0,C 180,E1 -30974.221,E2 -30974.221} C_VEL
LIN {X 0,Y 48.232,Z 309.101,A -85,B 0,C 180,E1 -30978.71,E2 -30978.71} C_VEL
LIN {X 0,Y 41.686,Z 311.721,A -85,B 0,C 180,E1 -30983.028,E2 -30983.028} C_VEL
LIN {X 0,Y 36.488,Z 313.386,A -85,B 0,C 180,E1 -30986.431,E2 -30986.431} C_VEL
LIN {X 0,Y 27.257,Z 315.502,A -85,B 0,C 180,E1 -30991.839,E2 -30991.839} C_VEL
LIN {X 0,Y 20.037,Z 316.626,A -85,B 0,C 180,E1 -30999.513,E2 -30999.513} C_VEL
LIN {X 0,Y 15.576,Z 317.193,A -85,B 0,C 180,E1 -31012.003,E2 -31012.003} C_VEL
LIN {X 0,Y 14.532,Z 317.321,A -85,B 0,C 180,E1 -31018.342,E2 -31018.342} C_VEL
LIN {X 0,Y 12.929,Z 317.593,A -85,B 0,C 180,E1 -31049.992,E2 -31049.992} C_VEL
LIN {X 0,Y 14.272,Z 317.353,A -85,B 0,C 180,E1 -31079.492,E2 -31079.492} C_VEL
LIN {X 0,Y 18.35,Z 316.725,A -85,B 0,C 180,E1 -31099.986,E2 -31099.986} C_VEL
LIN {X 0,Y 23.806,Z 315.708,A -85,B 0,C 180,E1 -31112.323,E2 -31112.323} C_VEL
LIN {X 0,Y 29.911,Z 314.287,A -85,B 0,C 180,E1 -31120.015,E2 -31120.015} C_VEL
LIN {X 0,Y 39.72,Z 311.327,A -85,B 0,C 180,E1 -31126.685,E2 -31126.685} C_VEL
LIN {X 0,Y 49.842,Z 307.331,A -85,B 0,C 180,E1 -31130.749,E2 -31130.749} C_VEL
LIN {X 0,Y 60.106,Z 302.193,A -85,B 0,C 180,E1 -31133.608,E2 -31133.608} C_VEL
LIN {X 0,Y 62.977,Z 300.38,A -85,B 0,C 180,E1 -31135.76,E2 -31135.76} C_VEL
LIN {X 0,Y 63.812,Z 299.661,A -85,B 0,C 180,E1 -31140,E2 -31140} C_VEL
LIN {X 0,Y 63.047,Z 300.074,A -85,B 0,C 180,E1 -31145.15,E2 -31145.15} C_VEL
LIN {X 0,Y 62.845,Z 300.228,A -85,B 0,C 180,E1 -31146.421,E2 -31146.421} C_VEL
LIN {X 0,Y 59.979,Z 301.935,A -85,B 0,C 180,E1 -31148.396,E2 -31148.396} C_VEL
LIN {X 0,Y 50.129,Z 306.798,A -85,B 0,C 180,E1 -31151.083,E2 -31151.083} C_VEL
LIN {X 0,Y 40.089,Z 310.731,A -85,B 0,C 180,E1 -31155.388,E2 -31155.388} C_VEL
LIN {X 0,Y 30.406,Z 313.63,A -85,B 0,C 180,E1 -31162.409,E2 -31162.409} C_VEL
LIN {X 0,Y 18.887,Z 315.991,A -85,B 0,C 180,E1 -31181.917,E2 -31181.917} C_VEL
LIN {X 0,Y 13.132,Z 316.81,A -85,B 0,C 180,E1 -31230.008,E2 -31230.008} C_VEL
LIN {X 0,Y 14.714,Z 316.613,A -85,B 0,C 180,E1 -31258.539,E2 -31258.539} C_VEL
LIN {X 0,Y 18.889,Z 316.026,A -85,B 0,C 180,E1 -31278.094,E2 -31278.094} C_VEL
LIN {X 0,Y 30.391,Z 313.7,A -85,B 0,C 180,E1 -31297.678,E2 -31297.678} C_VEL
LIN {X 0,Y 40.073,Z 310.83,A -85,B 0,C 180,E1 -31304.718,E2 -31304.718} C_VEL
LIN {X 0,Y 50.123,Z 306.93,A -85,B 0,C 180,E1 -31308.975,E2 -31308.975} C_VEL
LIN {X 0,Y 60.013,Z 302.079,A -85,B 0,C 180,E1 -31311.678,E2 -31311.678} C_VEL
LIN {X 0,Y 62.93,Z 300.362,A -85,B 0,C 180,E1 -31313.588,E2 -31313.588} C_VEL
LIN {X 0,Y 63.394,Z 300.034,A -85,B 0,C 180,E1 -31316.182,E2 -31316.182} C_VEL
LIN {X 0,Y 63.868,Z 299.808,A -85,B 0,C 180,E1 -31320,E2 -31320} C_VEL
LIN {X 0,Y 63.021,Z 300.538,A -85,B 0,C 180,E1 -31324.324,E2 -31324.324} C_VEL
LIN {X 0,Y 60.11,Z 302.354,A -85,B 0,C 180,E1 -31326.396,E2 -31326.396} C_VEL
LIN {X 0,Y 49.847,Z 307.456,A -85,B 0,C 180,E1 -31329.259,E2 -31329.259} C_VEL
LIN {X 0,Y 38.757,Z 311.731,A -85,B 0,C 180,E1 -31333.816,E2 -31333.816} C_VEL
LIN {X 0,Y 29.915,Z 314.352,A -85,B 0,C 180,E1 -31339.984,E2 -31339.984} C_VEL
LIN {X 0,Y 23.809,Z 315.753,A -85,B 0,C 180,E1 -31347.673,E2 -31347.673} C_VEL
LIN {X 0,Y 14.532,Z 317.321,A -85,B 0,C 180,E1 -31378.342,E2 -31378.342} C_VEL
LIN {X 0,Y 12.843,Z 317.572,A -85,B 0,C 180,E1 -31393.19,E2 -31393.19} C_VEL
LIN {X 0,Y 11.168,Z 317.636,A -85,B 0,C 180,E1 -31420.614,E2 -31420.614} C_VEL
LIN {X 0,Y 13.452,Z 317.001,A -85,B 0,C 180,E1 -31467.467,E2 -31467.467} C_VEL
LIN {X 0,Y 19.385,Z 315.894,A -85,B 0,C 180,E1 -31486.638,E2 -31486.638} C_VEL
LIN {X 0,Y 23.044,Z 315.157,A -85,B 0,C 180,E1 -31490.719,E2 -31490.719} C_VEL
LIN {X 0,Y 28.28,Z 314.072,A -85,B 0,C 180,E1 -31493.718,E2 -31493.718} C_VEL
LIN {X 0,Y 38.705,Z 311.113,A -85,B 0,C 180,E1 -31497.006,E2 -31497.006} C_VEL
LIN {X 0,Y 51.683,Z 305.986,A -85,B 0,C 180,E1 -31499.382,E2 -31499.382} C_VEL
LIN {X 0,Y 56.222,Z 303.803,A -85,B 0,C 180,E1 -31500,E2 -31500} C_VEL
LIN {X 0,Y 57.346,Z 303.193,A -85,B 0,C 180,E1 -31501.267,E2 -31501.267} C_VEL
LIN {X 0,Y 56.255,Z 303.744,A -85,B 0,C 180,E1 -31501.966,E2 -31501.966} C_VEL
LIN {X 0,Y 45.768,Z 308.428,A -85,B 0,C 180,E1 -31503.553,E2 -31503.553} C_VEL
LIN {X 0,Y 35.351,Z 312.001,A -85,B 0,C 180,E1 -31506.295,E2 -31506.295} C_VEL
LIN {X 0,Y 28.467,Z 313.844,A -85,B 0,C 180,E1 -31509.076,E2 -31509.076} C_VEL
LIN {X 0,Y 15.097,Z 316.204,A -85,B 0,C 180,E1 -31521.423,E2 -31521.423} C_VEL
LIN {X 0,Y 6.033,Z 317.023,A -85,B 0,C 180,E1 -31590.016,E2 -31590.016} C_VEL
LIN {X 0,Y 9.133,Z 316.826,A -85,B 0,C 180,E1 -31640.324,E2 -31640.324} C_VEL
LIN {X 0,Y 15.1,Z 316.238,A -85,B 0,C 180,E1 -31658.59,E2 -31658.59} C_VEL
LIN {X 0,Y 28.46,Z 313.913,A -85,B 0,C 180,E1 -31671.056,E2 -31671.056} C_VEL
LIN {X 0,Y 38.81,Z 311.042,A -85,B 0,C 180,E1 -31674.89,E2 -31674.89} C_VEL
LIN {X 0,Y 49.261,Z 307.142,A -85,B 0,C 180,E1 -31677.09,E2 -31677.09} C_VEL
LIN {X 0,Y 56.257,Z 303.907,A -85,B 0,C 180,E1 -31678.082,E2 -31678.082} C_VEL
LIN {X 0,Y 57.46,Z 303.303,A -85,B 0,C 180,E1 -31679.061,E2 -31679.061} C_VEL
LIN {X 0,Y 56.225,Z 303.963,A -85,B 0,C 180,E1 -31680,E2 -31680} C_VEL
LIN {X 0,Y 45.7,Z 308.677,A -85,B 0,C 180,E1 -31681.556,E2 -31681.556} C_VEL
LIN {X 0,Y 35.223,Z 312.28,A -85,B 0,C 180,E1 -31683.894,E2 -31683.894} C_VEL
LIN {X 0,Y 28.283,Z 314.138,A -85,B 0,C 180,E1 -31686.282,E2 -31686.282} C_VEL
LIN {X 0,Y 14.817,Z 316.544,A -85,B 0,C 180,E1 -31698.427,E2 -31698.427} C_VEL
LIN {X 0,Y 8.812,Z 317.16,A -85,B 0,C 180,E1 -31717.083,E2 -31717.083} C_VEL
LIN {X 0,Y 5.824,Z 317.379,A -85,B 0,C 180,E1 -31769.983,E2 -31769.983} C_VEL
LIN {X 0,Y 8.809,Z 317.14,A -85,B 0,C 180,E1 -31822.904,E2 -31822.904} C_VEL
LIN {X 0,Y 14.814,Z 316.511,A -85,B 0,C 180,E1 -31841.569,E2 -31841.569} C_VEL
LIN {X 0,Y 23.044,Z 315.157,A -85,B 0,C 180,E1 -31850.719,E2 -31850.719} C_VEL
LIN {X 0,Y 25.354,Z 317.118,A -85,B 0,C 180,E1 -31852.2,E2 -31852.2} C_VEL
LIN {X 0,Y 25.354,Z 600,A -85,B 0,C 180,E1 -31852.2,E2 -31852.2} C_VEL
LIN {X 0,Y 25.354,Z 600,A -85,B 0,C 180,E1 -31852.2,E2 -31852.2}

QRS_NEXT_CUT()

QRS_NEXT()
QRS_HOME()

END
